FUNCTION_BLOCK relaxPistons
VAR_INPUT
END_VAR
VAR_OUTPUT
END_VAR
VAR
END_VAR

IF I_bRightLiftBottom THEN
	O_bRightLiftDown:=FALSE;
END_IF

IF  I_bRightLiftUp THEN
	O_bRightLiftUp:=FALSE;
END_IF

IF I_bLeftLiftBottom THEN
	O_bLeftLiftDown:=FALSE;
END_IF

IF  I_bLeftLiftUp THEN
	O_bLeftLiftUp:=FALSE;
END_IF

END_FUNCTION_BLOCK

(* stored: Version 1.1.0.1, ProductVersion 3.1.4018.2
   POU relaxPistons: Id {c9fadeb7-dc15-454c-b494-4cd261c8c5e7}, SpecialFunc None *)
